FUNCTION_BLOCK ABSTRACT RunningToHaltedProgramTransition EXTENDS ProgramTransition

{attribute 'monitoring' := 'call'}
{attribute 'OPC.UA.DA.Property' := '1'}
{attribute 'OPC.UA.DA.Access' := '1'}
PROPERTY FINAL Cause : STRING
GET
Cause := 'Halt';
END_GET
END_PROPERTY

{attribute 'monitoring' := 'call'}
{attribute 'OPC.UA.DA.Property' := '1'}
{attribute 'OPC.UA.DA.Access' := '1'}
PROPERTY FINAL FromState : STRING
GET
FromState := 'Running';
END_GET
END_PROPERTY

{attribute 'monitoring' := 'call'}
{attribute 'OPC.UA.DA.Property' := '1'}
{attribute 'OPC.UA.DA.Access' := '1'}
PROPERTY FINAL Name : STRING
GET
Name := 'RunningToHalted';
END_GET
END_PROPERTY

{attribute 'monitoring' := 'call'}
{attribute 'OPC.UA.DA.Property' := '1'}
{attribute 'OPC.UA.DA.Access' := '1'}
PROPERTY FINAL ToState : STRING
GET
ToState := 'Halted';
END_GET
END_PROPERTY

END_FUNCTION_BLOCK

(* stored: Version 1.1.0.1
   POU RunningToHaltedProgramTransition: Id {8a6734b4-3b9e-42db-8f8f-8ed9038de12d}, SpecialFunc None
   Property Cause: Id {9ce43ec7-8a88-4a6a-ae50-c578da3da785}
   Get Get: Id {f71d1651-79fa-49fd-836b-b1342ffcf471}
   Property FromState: Id {5920b324-7b3d-4765-b17f-c5375d0a1800}
   Get Get: Id {42e3645d-6610-4221-ad79-fe44ccb91ee8}
   Property Name: Id {5bf2e8bf-beb8-4504-862f-50899bc78b22}
   Get Get: Id {09de0d78-62ca-45fd-ae9b-4b4efcc46fae}
   Property ToState: Id {bc3b59ab-11a2-47c7-9789-b60431e7b912}
   Get Get: Id {a99a9f8e-182e-4180-b2e1-268fb173d262} *)
